TYPE st_Pump_Output :
STRUCT
	On : BOOL;
END_STRUCT
END_TYPE

(* stored: Version 1.1.0.1, ProductVersion 3.1.4024.9
   DUT st_Pump_Output: Id {feb95ab5-d4b0-4603-acd9-02cd62d0bbd8} *)
